(* PLC project TEST.project, CODESYS CODESYS V3.5 SP3 Patch 7 *)
(* stored: creationDateTime 2013-12-18T19:32:28.4147223, modificationDateTime 2013-12-18T18:56:49.0513577 *)

FUNCTION_BLOCK Motor
  VAR
    Signal : INT;
    AUS : INT;
  END_VAR

INITIAL_STEP Motor AUS:
END_STEP
TRANSITION FROM Motor AUS TO Motor dreht links
  := Signal 1;
END_TRANSITION
TRANSITION FROM Motor AUS TO Motor dreht rechts
  := Signal 2;
END_TRANSITION
STEP Motor dreht links:
END_STEP
TRANSITION FROM Motor dreht links TO Init
  := Signal AUS;
END_TRANSITION
STEP Motor dreht rechts:
END_STEP
TRANSITION FROM Motor dreht rechts TO Init
  := Trans1;
END_TRANSITION
END_FUNCTION_BLOCK
